FUNCTION_BLOCK FB_HistoryUpdate_LREAL
VAR_INPUT
	bSample			: BOOL := TRUE; //Set True if data should be sampled; set FALSE if sampling should be stopped.
	bStop			: BOOL; // set TRUE if nodes should be released
	nConnectionHdl	: DWORD;
	nNamespaceIndex	: UINT;
	sNodeIdentifier	: STRING(MAX_STRING_LENGTH);
	pValue			: PVOID;
END_VAR
VAR_OUTPUT
	bBusy			: BOOL;
	bError			: BOOL;
	nErrorID		: DWORD;
	nNodeHdl		: DWORD;
END_VAR

VAR CONSTANT
	cBufferSize		: UINT := 1000;
	cValueSize		: UINT := SIZEOF(LREAL);
END_VAR
VAR
	// state machine declarations 
	RisingEdgeStart			: R_TRIG;
	nState					: INT := 0;

	// Declarations for UA_NodeGetHandle
	fbUANodeGetHandle		: UA_NodeGetHandle;
	NodeID					: ST_UANodeID := (eIdentifierType 	:= eUAIdentifierType_String);
	
	// Declarations for UA_HistoryUpdate
	fbUAHistoryUpdate		: UA_HistoryUpdate;
	aDataValues				: ARRAY [1..cBufferSize] OF UAHADataValue(ValueSize:=cValueSize);
	aValueErrorIDs			: ARRAY [1..cBufferSize] OF DWORD;
	nCounter				: UINT := 1;
	
	// Declarations for UA_NodeReleaseHandle
	fbUANodeReleaseHandle	: UA_NodeReleaseHandle;
END_VAR

RisingEdgeStart(CLK:=bSample);

CASE nState OF
0: //Idle	
	IF RisingEdgeStart.Q THEN
		bError := FALSE;
		nErrorID := 0;
		nCounter := 1;
		
		NodeID.nNamespaceIndex 	:= nNamespaceIndex;
		NodeID.sIdentifier		:= sNodeIdentifier;
		
		fbUANodeGetHandle(	Execute 			:= TRUE,
							ConnectionHdl 		:= nConnectionHdl,
							NodeID 				:= NodeID,
							Busy				=> bBusy );	
		nState := 1;	
	END_IF
	
1: //Get Node Handle
	fbUANodeGetHandle(Execute := FALSE, NodeHdl=>nNodeHdl, Busy=>bBusy );
	IF NOT fbUANodeGetHandle.Busy THEN
		IF NOT fbUANodeGetHandle.Error THEN
			nCounter		:= 1;
			nState 			:= 2;
		ELSE
			bError  		:= TRUE;
			nErrorID 		:= fbUANodeGetHandle.ErrorID;
			nState 			:= 666; //error state
		END_IF
	END_IF
	
2: //UA_HistoryUpdate
	IF bSample THEN
		aDataValues[nCounter].Value			 	:= pValue;
		aDataValues[nCounter].StatusCode 		:= UAHAUpdateStatusCode.HistorianRaw;
		aDataValues[nCounter].ServerTimeStamp 	:= F_GetSystemTime();
		aDataValues[nCounter].SourceTimeStamp 	:= aDataValues[nCounter].ServerTimeStamp;	
		nCounter := nCounter + 1;

		IF nCounter > cBufferSize THEN
			fbUAHistoryUpdate.Execute := TRUE;
			nCounter := 1;
		END_IF
	END_IF
	
	fbUAHistoryUpdate(	Execute 		:= , //already set above
						ConnectionHdl 	:= nConnectionHdl,
						NodeHdl 		:= nNodeHdl,
						PerformInsert 	:= TRUE,
						PerformReplace 	:= FALSE,
						DataValueCount 	:= cBufferSize,
						DataValues	 	:= aDataValues,
						ValueErrorIDs 	:= aValueErrorIDs,
						Busy			=> bBusy );
						
	IF NOT fbUAHistoryUpdate.Busy THEN
		IF NOT fbUAHistoryUpdate.Error THEN
			IF bStop THEN
				nState := 3; //Release Node Handle
			END_IF
		ELSE
			bError 			:= TRUE;
			nErrorID 		:= fbUAHistoryUpdate.ErrorID;
			nState 			:= 666; //error state
		END_IF
		fbUAHistoryUpdate(	Execute			:= FALSE, 			
							DataValues	 	:= aDataValues,
							ValueErrorIDs 	:= aValueErrorIDs,
							Busy			=> bBusy );
	END_IF
	
3: //Release Node Handle
	fbUANodeReleaseHandle(	Execute 		:= TRUE,
							ConnectionHdl 	:= nConnectionHdl,
							NodeHdl 		:= nNodeHdl,
							Busy			=> bBusy );
		
	IF NOT fbUANodeReleaseHandle.Busy THEN
		IF NOT fbUANodeReleaseHandle.Error THEN
			nState		:= 0;
			nNodeHdl	:= 0;
		ELSE
			bError 		:= TRUE;
			nErrorID 	:= fbUANodeReleaseHandle.ErrorID;
			nState 		:= 666; //error state
		END_IF
		fbUANodeReleaseHandle(Execute := FALSE, Busy => bBusy );
	END_IF	
	
666: //error state	
	
END_CASE

END_FUNCTION_BLOCK

(* stored: Version 1.1.0.1, ProductVersion 3.1.4024.9
   POU FB_HistoryUpdate_LREAL: Id {ccca5662-2355-453d-8dde-518ed392a616}, SpecialFunc None *)
